DATA_BLOCK "STATION"
{ S7_Optimized_Access := 'TRUE' }
VERSION : 0.1
NON_RETAIN
   VAR RETAIN
      Count : UInt;
      Station { S7_SetPoint := 'False'} : Array["STATION_MIN".."STATION_MAX"] of "LGR_Station_Para";
   END_VAR


BEGIN
   Count := 32;

END_DATA_BLOCK

